// TwinCAT 3 PLC project PLC1
// ProgramVersion: 3.1.4023.0
// libraries:
//   Tc2_Standard, * (Beckhoff Automation GmbH)
//   Tc2_System, * (Beckhoff Automation GmbH)
//   Tc3_Module, * (Beckhoff Automation GmbH)
//   VisuDialogs, * (System)
//   VisuSymbols,3.5.10.0,System
// project tree:
//   DUTs/ ST_HOLES.TcDUT
//   / GlobalTextList.TcGTLO, PlcTask.TcTTO, Visualization Manager.TcVMO (not stored)
//   GVLs/ MAINVARS.TcGVL
//   POUs/ MAIN.TcPOU, HOMING.TcPOU
//   VISUs/ HMI1.TcVIS
// real-time tasks:
//   TASK PlcTask: cycle T#1ms, priority 20, ADS port 350
// I/O:
//   DEVICE Device 1 (EtherCAT), AmsNetId 192.168.1.8.2.1
//     Box 2 (EasyCAT 32+32 rev 1) [ Generic 32+32 bytes rev 1 ]
// variable links:
//   PLC1/PLC1 Instance <-> Device 1 (EtherCAT)/Box 2 (EasyCAT 32+32 rev 1)
//     PlcTask Inputs/MAINVARS.BitIn0 <-> Inputs/Byte6
//     PlcTask Inputs/MAINVARS.BitIn{1..7} <-> Inputs/Byte6 @bit {1..7}  (7 links)
//     PlcTask Outputs/MAINVARS.BitOut0 <-> Outputs/Byte0
//     PlcTask Outputs/MAINVARS.BitOut8 <-> Outputs/Byte1
//     PlcTask Outputs/MAINVARS.BitOut1 <-> Outputs/Byte0 @bit 1
//     PlcTask Outputs/MAINVARS.BitOut2 <-> Outputs/Byte0 @bit 2
//     PlcTask Outputs/MAINVARS.BitOut3 <-> Outputs/Byte0 @bit 3
//     PlcTask Outputs/MAINVARS.BitOut4 <-> Outputs/Byte0 @bit 4
//     PlcTask Outputs/MAINVARS.BitOut5 <-> Outputs/Byte0 @bit 5
//     PlcTask Outputs/MAINVARS.BitOut6 <-> Outputs/Byte0 @bit 6
//     PlcTask Outputs/MAINVARS.BitOut7 <-> Outputs/Byte0 @bit 7
//     PlcTask Outputs/MAINVARS.BitOut9 <-> Outputs/Byte1 @bit 1

CONFIGURATION PLC1
    RESOURCE PLC ON TwinCAT3
        TASK PlcTask(INTERVAL := T#1ms, PRIORITY := 20);
        PROGRAM MAIN WITH PlcTask : MAIN;
    END_RESOURCE
END_CONFIGURATION

// ---- DUTs/ST_HOLES.TcDUT
TYPE ST_HOLES :
STRUCT
	rX : REAL;
	rY : REAL;
END_STRUCT
END_TYPE

// ---- GVLs/MAINVARS.TcGVL
{attribute 'qualified_only'}
VAR_GLOBAL
	Ana0 AT %I* : INT;
	Ana1 AT %I* : INT;
	
	BitOut0 AT %Q* : BOOL := TRUE; // Enable motor 1
	BitOut1 AT %Q* : BOOL := FALSE; // Direction motor 1 
	BitOut2 AT %Q* : BOOL := FALSE; // Step motor 1
	BitOut3 AT %Q* : BOOL := FALSE;  // BUSY motor 1
	BitOut4 AT %Q* : BOOL := FALSE; // Alarm motor 1
	
	BitOut5 AT %Q* : BOOL := TRUE;  // Enable motor 2 
	BitOut6 AT %Q* : BOOL := FALSE; // Direction  motor 2
	BitOut7 AT %Q* : BOOL := FALSE; // Step Motor 2
	BitOut8 AT %Q* : BOOL := FALSE; //  Busy motor 2
	BitOut9 AT %Q* : BOOL := FALSE; // Alamrm motor 2 
	
	BitOut10 AT %I* : REAL := 0.0;  //  SetSpeed 1
	BitOut11 AT %I* : REAL := 0.0;  //  SetSpeed 2
	BitOut12 AT %I* : REAL := 0.0;  //  ToPosition 1
	BitOut13 AT %I* : REAL := 0.0;  //  ToPosition 2
 
	
	BitIn0 AT %I* : BOOL := FALSE;  // Limit 1/1
	BitIn1 AT %I* : BOOL := FALSE;  // Limit 1/2
	BitIn2 AT %I* : BOOL := FALSE;	// Limit 2/1
	BitIn3 AT %I* : BOOL := FALSE;  // Limit 2/2
	BitIn4 AT %I* : BOOL := FALSE;	// Busy M1
	BitIn5 AT %I* : BOOL := FALSE;  // Busy M1
	BitIn6 AT %I* : BOOL := FALSE;	// Alarm M1
	BitIn7 AT %I* : BOOL := FALSE;  // Alarm M2
	BitIn8 AT %I* : BOOL := FALSE;  // M1 IsHomed
	BitIn9 AT %I* : BOOL := FALSE;  // M2 IsHomed

	

	GlobalAlarm: BOOL := 0;
	EmergencyStop: BOOL := 0;
	AlarmMessage: STRING := 'No alarm';
	ContToNextStage: INT := 0;;
	MachineState: INT := 0;
	PreviousMachineState: INT;
	Start: BOOL := FALSE;
	heartbeat : BYTE;
	
END_VAR

// ---- POUs/MAIN.TcPOU
PROGRAM MAIN
VAR
	
	stHoles : ST_HOLES;
	i : DINT;
	aHoles : ARRAY [0..NUM_HOLES] OF ST_HOLES;
	
END_VAR
VAR CONSTANT
	NUM_HOLES : DINT := 2;
END_VAR

// Check MAchineState and Alarms
// Check for alarms and act on it if necessairy.
MAINVARS.heartbeat := MAINVARS.heartbeat + 1;

//MAINVARS.BitOut0 := MAINVARS.heartbeat MOD 2 = 0;
//MAINVARS.BitOut1 := MAINVARS.heartbeat MOD 4 = 0;
//MAINVARS.BitOut2 := MAINVARS.heartbeat MOD 8 = 0;
//MAINVARS.BitOut3 := MAINVARS.heartbeat MOD 16 = 0;


// If there's no globalalarm then proceed normally;
IF MAINVARS.GlobalAlarm = FALSE THEN
	CASE MAINVARS.MachineState  OF
		0:
			// Do Nothing Machine is in rest mode
			MAINVARS.BitOut0 := TRUE; // Disabled
			MAINVARS.BitOut1 := FALSE; // CW / CCW
			MAINVARS.BitOut2 := FALSE; // Disabled
			MAINVARS.BitOut3 := FALSE; // !Enabled
			MAINVARS.BitOut4 := FALSE; // !Enabled
			
			MAINVARS.BitOut5 := TRUE; // Disabled
			MAINVARS.BitOut6 := FALSE; // CW / CCW
			MAINVARS.BitOut7 := FALSE; // Disabled
			MAINVARS.BitOut8 := FALSE; // !Enabled
			MAINVARS.BitOut9 := FALSE; // !Enabled
			
			MAINVARS.MachineState := 0;
			MAINVARS.AlarmMessage := 'Ready';
			IF(MAINVARS.Start = TRUE AND MAINVARS.PreviousMachineState <> 20) THEN
				// Set previous and current machine state for next step	
				MAINVARS.PreviousMachineState := 0;
				MAINVARS.MachineState := 10;
			END_IF
		10: 
			// Home X
			MAINVARS.AlarmMessage := 'Homing X';
			REPEAT
				MAINVARS.BitOut0 := FALSE; // !Enabled
				MAINVARS.BitOut1 := TRUE; // !Enabled
				MAINVARS.BitOut2 := TRUE; // !Enabled
				MAINVARS.BitOut3 := TRUE; // !Enabled
				MAINVARS.BitIn8 := FALSE;   // IsHomed
			UNTIL 
				MAINVARS.BitIn0 = FALSE
			END_REPEAT;

				
			
//			IF MAINVARS.BitIn0 <> FALSE  THEN
//				MAINVARS.BitOut0 := FALSE; // !Enabled
//				MAINVARS.BitOut1 := TRUE; // !Enabled
//				MAINVARS.BitOut2 := TRUE; // !Enabled
//				MAINVARS.BitOut3 := TRUE; // !Enabled
//				MAINVARS.BitIn8 := FALSE;   // IsHomed
//			ELSE 
//				MAINVARS.BitOut0 := TRUE; // Disabled M1
//				MAINVARS.BitOut1 := TRUE; // M1 CW
//				MAINVARS.BitOut2 := FALSE; // NO STEPS
//				MAINVARS.BitOut3 := FALSE; // NOT BUSY
//				MAINVARS.BitIn8 := TRUE;   // IsHomed
//				MAINVARS.PreviousMachineState := 10;
//				MAINVARS.MachineState := 20;
//			END_IF
			
		
			
		20:
			/// Home Y
			MAINVARS.AlarmMessage := 'Homing Y';
			
			// Set previous and current machine state for next step	
			
			
			IF MAINVARS.BitIn0 <> FALSE  THEN
				MAINVARS.BitOut5 := FALSE; // !Enabled
				MAINVARS.BitOut6 := TRUE; // !Enabled
				MAINVARS.BitOut7 := TRUE; // !Enabled
				MAINVARS.BitOut8 := TRUE; // !Enabled
				MAINVARS.BitIn9 := FALSE;   // IsHomed
			ELSE 
				MAINVARS.BitOut5 := TRUE; // Disabled M1
				MAINVARS.BitOut6 := TRUE; // M1 CW
				MAINVARS.BitOut7 := FALSE; // NO STEPS
				MAINVARS.BitOut8 := FALSE; // NOT BUSY
				MAINVARS.BitIn9 := TRUE;   // IsHomed
				MAINVARS.Start := FALSE;
				MAINVARS.PreviousMachineState := 20;
				MAINVARS.MachineState := 0;
			END_IF
			
			
		
	   999: // Handle error;
			IF MAINVARS.GlobalAlarm = TRUE THEN
				MAINVARS.EmergencyStop := 1;
				MAINVARS.AlarmMessage := 'Alarm: ';
				MAINVARS.ContToNextStage := 0;	
				// Depending on the machine state take action.
				
			END_IF
			
			  
	END_CASE
END_IF

END_PROGRAM

// ---- POUs/HOMING.TcPOU
FUNCTION HOMING : BOOL
VAR_INPUT
END_VAR
VAR
END_VAR

END_FUNCTION

// ---- GlobalTextList.TcGTLO
TEXTLIST GlobalTextList
  722 = '+'
  880 = '-'
  843 = 'Alarm'
  145 = 'Home'
  135 = 'Motor 1 Run'
  310 = 'Motor 2 Run'
  152 = 'Motor enabled'
  942 = 'Motor1 Enabled'
  556 = 'Out 4 HIGH/LOW'
  318 = 'Ready'
  596 = 'Stage: %s'
  601 = 'Start'
  37 = 'Status: %s'
  505 = 'Stop'
END_TEXTLIST

// ---- VISUs/HMI1.TcVIS
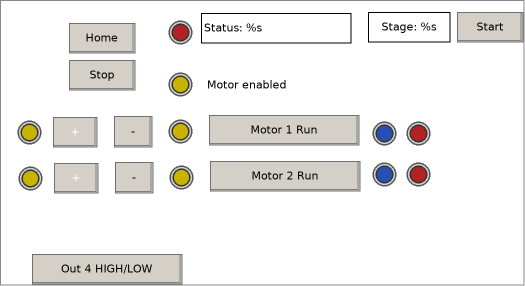
VISUALIZATION HMI1  // 525x286
    Button (53,117 44x30), "+"
        OnMouseClick: execute {
            MAINVARS.BitOut0 := FALSE;
            MAINVARS.BitOut1 := TRUE;
            MAINVARS.BitOut2 := TRUE;
        }
        OnMouseLeave: execute { MAINVARS.BitOut0 := TRUE; }
    Button (114,116 38x31), "-"
        OnMouseClick: execute {
            MAINVARS.BitOut0 := FALSE;
            MAINVARS.BitOut1 := FALSE;
            MAINVARS.BitOut2 := TRUE;
        }
        OnMouseLeave: execute { MAINVARS.BitOut0 := TRUE; }
    Button (69,23 66x30), "Home"
    Lamp1 (16,119 27x27), variable: MAINVARS.BitOut1 = TRUE;, style: Lamp-Lamp1-Yellow
    Lamp1 (167,71 27x27), variable: MAINVARS.BitOut0 = FALSE OR MAINVARS.BitOut5 = FALSE;, style: Lamp-Lamp1-Yellow
    Label (204,70 94x30), "Motor enabled"
    Lamp1 (167,118 27x27), variable: MAINVARS.BitOut1 = FALSE;, style: Lamp-Lamp1-Yellow
    Lamp1 (167,19 27x27), variable: MAINVARS.GlobalAlarm, style: Lamp-Lamp1-Red
    Rectangle (201,13 150x30), "Status: %s", text variable: MAINVARS.AlarmMessage
    Button (69,60 66x30), "Stop"
        OnMouseClick: execute {
            MAINVARS.BitOut0 := TRUE;
            MAINVARS.BitOut2 := FALSE;
            MAINVARS.Start := FALSE;
            MAINVARS.AlarmMessage := 'Stopped';
            MAINVARS.MachineState := 0;
            MAINVARS.PreviousMachineState := 0;
        }
    Rectangle (368,12 82x30), "Stage: %s", text variable: MAINVARS.MachineState
    Button (457,12 66x30), "Start"
        OnMouseClick: toggle MAINVARS.Start
    Button (209,115 150x30), "Motor 1 Run"
        OnMouseClick: execute { MAINVARS.BitOut2 := TRUE; }
        OnMouseUp: execute { MAINVARS.BitOut2 := FALSE; }
    Button (32,254 150x30), "Out 4 HIGH/LOW"
        toggle MAINVARS.BitOut3
    Button (54,163 44x30), "+"
        OnMouseClick: execute {
            MAINVARS.BitOut5 := FALSE;
            MAINVARS.BitOut6 := TRUE;
            MAINVARS.BitOut7 := TRUE;
        }
        OnMouseLeave: execute { MAINVARS.BitOut5 := TRUE; }
    Button (115,162 38x31), "-"
        OnMouseClick: execute {
            MAINVARS.BitOut5 := FALSE;
            MAINVARS.BitOut6 := FALSE;
            MAINVARS.BitOut7 := TRUE;
        }
        OnMouseLeave: execute { MAINVARS.BitOut5 := TRUE; }
    Lamp1 (17,165 27x27), variable: MAINVARS.BitOut6 = TRUE;, style: Lamp-Lamp1-Yellow
    Lamp1 (168,164 27x27), variable: MAINVARS.BitOut6 = FALSE;, style: Lamp-Lamp1-Yellow
    Button (210,161 150x30), "Motor 2 Run"
        OnMouseClick: execute { MAINVARS.BitOut2 := TRUE; }
        OnMouseUp: execute { MAINVARS.BitOut2 := FALSE; }
    Lamp1 (371,120 27x27), variable: MAINVARS.BitIn4 = FALSE, style: Lamp-Lamp1-Blue
    Lamp1 (371,161 27x27), variable: MAINVARS.BitIn5 = FALSE, style: Lamp-Lamp1-Blue
    Lamp1 (405,120 27x27), variable: MAINVARS.BitIn0 = FALSE, style: Lamp-Lamp1-Red
    Lamp1 (405,161 27x27), variable: MAINVARS.BitIn2 = FALSE, style: Lamp-Lamp1-Red
END_VISUALIZATION
